// TIA Portal V19 export
DATA_BLOCK "Setpoints_Polygon"   // DB115
{ S7_Optimized_Access := 'TRUE' }
// stored: AutoNumber false, MemoryReserve 0
   VAR RETAIN
      TT0941_CondenseHigh : Real := 70.0;   // TT0941 Condensate Temperature Fault High
      TT0941_CondenseLow : Real := 0.0;   // TT0941 Condensate Temperature Fault Low
      TT0940_Low_Prod : Real := 110.0;   // TT0940 Low Temperature
      TT0940_Low_SIP : Real := 125.0;   // TT0940 Low Temperature
      TT0941_Low_SIP : Real := 125.0;   // TT0941 Low Temperature
      CT0931_High : Real := 100.0;   // CT0931 High Conductivity - Suspect product in Condensate
      EOL_Barrier_Low_Prod : Real := 110.0;   // TT1040 or TT1041 Low Temperature during Production
      EOL_Barrier_Low_SIP : Real := 125.0;   // TT1040 or TT1041 Low Temperature during Sterilising
      PG_F2_ProdAtFillerSet : Real := 2000.0;   // CTX2274 Minimum Conductivity of Product in microSeimens
      PG_F2_ProdAtFillerReset : Real := 1500.0;   // CTX2274 Maximum Conductivity of Potable Water in microSeimens
      PG_F2_ProdAtFillerDlyOn : S5Time := S5T#5S;   // Product at Filler 2 Delay On Time.
      PG_F2_ProdAtFillerDlyOff : S5Time := S5T#1S;   // Product at Filler 2 Delay Off Time.
   END_VAR
BEGIN
END_DATA_BLOCK
